// TIA Portal V19 export
VAR_GLOBAL   // PLC tag table "Digitale Eingänge"
   "E_Si_24VDC_CM01.MM01" AT %I0.0 : Bool;   // LSS 24 V OK Deckelzylinder links CM01.MM01
   "E_Si_24VDC_CM01.MM02" AT %I0.1 : Bool;   // LSS 24 V OK Deckelzylinder rechts CM01.MM02
   "E_Si_24VDC_CM02.MM03" AT %I0.2 : Bool;   // LSS 24 V OK Deckelzylinder links CM02.MM03
   "E_Si_24VDC_CM02.MM04" AT %I0.3 : Bool;   // LSS 24 V OK Deckelzylinder rechts CM02.MM04
   "R E 0.4" AT %I0.4 : Bool;
   "R E 0.5" AT %I0.5 : Bool;
   "R E 0.6" AT %I0.6 : Bool;
   E_RM_NH_Dkl AT %I0.7 : Bool;   // Rückmeldung Nothalt Deckelzylinder CM01.MM01 ... CM02.MM04
   E_Dkl_li_auf_CM01 AT %I1.0 : Bool;   // Deckel links offen int Säure CM01
   E_Dkl_li_zu_CM01 AT %I1.1 : Bool;   // Deckel links geschlossen int Säure CM01
   E_Dkl_re_auf_CM01 AT %I1.2 : Bool;   // Deckel rechts offen int Säure CM01
   E_Dkl_re_zu_CM01 AT %I1.3 : Bool;   // Deckel rechts geschlossen int Säure CM01
   "E_S_Dkl_li_auf_CM01.BG01" AT %I1.4 : Bool;   // Stellrückmeldung Deckel links offen ext CM01.BG01
   "E_S_Dkl_li_zu_CM01.BG02" AT %I1.5 : Bool;   // Stellrückmeldung Deckel links geschlossen ext CM01.BG02
   "E_S_Dkl_re_auf_CM01.BG03" AT %I1.6 : Bool;   // Stellrückmeldung Deckel rechts offen ext CM01.BG03
   "E_S_Dkl_re_zu_CM01.BG04" AT %I1.7 : Bool;   // Stellrückmeldung Deckel rechts geschlossen ext CM01.BG04
   "E_Niv_UeL_CM01.BL01" AT %I2.0 : Bool;   // Überfüllsensor Max-Max Säure CM01 CM01.BL01
   "E_Niv_Max_CM01.BL02" AT %I2.1 : Bool;   // Füllstandssensor Max Säure CM01 CM01.BL02
   "E_Niv_Min_CM01.BL03" AT %I2.2 : Bool;   // Füllstandssensor Min Säure CM01 CM01.BL03
   "E_Niv_TLS_CM01.BL04" AT %I2.3 : Bool;   // Trockenlaufschutz Min Min Säure CM01 CM01.BL04
   "E_SRM_CM01.QM25_zu" AT %I2.4 : Bool;   // Stellrückmeldung ZU Eingang Saugleitung Umwälzpumpe GP02 CM01.BG-QM25
   "E_SRM_CM01.QM18_zu" AT %I2.5 : Bool;   // Stellrückmeldung ZU Eingang Saugleitung Filterpumpe GP01 CM01.BG-QM18
   "E_SRM_CM01.QM19_zu" AT %I2.6 : Bool;   // Stellrückmeldung ZU Eingang Spülleitung Filterpumpe GP01 CM01.BG-QM19
   "E_SRM_CM01.QM20_zu" AT %I2.7 : Bool;   // Stellrückmeldung ZU Eingang Spülleitung Umwälzpumpe GP02 CM01.BG-QM20
   "E_SRM_CM01.QM26_zu" AT %I3.0 : Bool;   // Stellrückmeldung ZU Ausgang Druckleitung Umwälzpumpe GP02 CM01.BG-QM26
   "E_SRM_CM01.QM27_zu" AT %I3.1 : Bool;   // Stellrückmeldung ZU Ausgang Spülleitung Umwälzpumpe GP02 zu Sammeltank CM01.BG-QM27
   "E_GW_LF_CM01.BN01" AT %I3.2 : Bool;   // Leitfähigkeit Bypass Filterpumpe CM01.BN01
   "E_GW_LF_CM01.BN02" AT %I3.3 : Bool;   // Leitfähigkeit Düsen Umwälzung CM01.BN02
   "E_GW_p_CM01.BP03" AT %I3.4 : Bool;   // Drucksensor Filterpumpe GP01 CM01.BP03
   "E_GW_p_CM01.BP04" AT %I5.2 : Bool;   // Drucksensor Umwälzpumpe GP02 CM01.BP04
   "R E 3.6" AT %I3.6 : Bool;
   "R E 3.7" AT %I3.7 : Bool;
   "E_SRM_HQ01.QM21_auf" AT %I4.0 : Bool;   // Stellrückmeldung AUF Eingang Säureleitung Filtereinheit HQ01 HQ01.QM21
   "R E4.1" AT %I4.1 : Bool;
   "E_S_FG_li_HQ01.BG07" AT %I4.2 : Bool;   // Positionssensor Filterdeckel links HQ01 HQ01.BG07
   "E_S_FG_re_HQ01.BG08" AT %I4.3 : Bool;   // Positionssensor Filterdeckel rechts HQ01 HQ01.BG08
   "E_SRM_HQ01.QM21_zu" AT %I4.4 : Bool;   // Stellrückmeldung ZU Eingang Säureleitung Filtereinheit HQ01 HQ01.BG-QM21
   "E_SRM_HQ01.QM23_zu" AT %I4.5 : Bool;   // Stellrückmeldung ZU Ausgang Säureleitung Filtereinheit HQ01 HQ01.BG-QM23
   "E_SRM_HQ01.QM24_zu" AT %I4.6 : Bool;   // Stellrückmeldung ZU Ausgang Spülleitung Filtereinheit HQ01 zu Sammeltank HQ01.BG-QM24
   "E_SRM_HQ01.LV01_zu" AT %I4.7 : Bool;   // Stellrückmeldung ZU Entlüftungs-/Überdruckventil Beutelfilter HQ01.BG-LV01
   "E_SRM_HQ01.QM22_zu" AT %I5.0 : Bool;   // Stellrückmeldung ZU Eingang Spülleitung Filtereinheit HQ01 CM01.BG-QM22
   "E_SRM_HQ01.QM23_auf" AT %I5.1 : Bool;   // Stellrückmeldung AUF Ausgang Säureleitung Filtereinheit HQ01 HQ01.BG-QM23
   "E_GW_p_HQ01.BP01" AT %I3.5 : Bool;   // Drucksensor Beutelfiltergehäuse HQ01 HQ01.BP01
   "E_GW_p_CM03.BP05" AT %I5.3 : Bool;   // Drucksensor Umwälzpumpe GP03 CM03.BP05
   "E_Niv_Min_CM03.BL06" AT %I5.4 : Bool;   // Füllstandssensor Min Spüle CM03 CM03.BL06
   "E_Niv_TLS_CM03.BL07" AT %I5.5 : Bool;   // Trockenlaufschutz Min Min Spüle CM03 CM03.BL07
   "E_SRM_CM03.QM33_zu" AT %I5.6 : Bool;   // Stellrückmeldung ZU Eingang Saugleitung Umwälzpumpe GP03 CM03.BG-QM33
   "E_SRM_CM03.QM34_zu" AT %I5.7 : Bool;   // Stellrückmeldung ZU Ausgang Druckleitung Umwälzpumpe GP03 CM03.BG-QM34
   E_Dkl_li_auf_CM02 AT %I6.0 : Bool;   // Deckel links offen int Säure CM02
   E_Dkl_li_zu_CM02 AT %I6.1 : Bool;   // Deckel links geschlossen int Säure CM02
   E_Dkl_re_auf_CM02 AT %I6.2 : Bool;   // Deckel rechts offen int Säure CM02
   E_Dkl_re_zu_CM02 AT %I6.3 : Bool;   // Deckel rechts geschlossen int Säure CM02
   "E_S_Dkl_li_auf_CM02.BG12" AT %I6.4 : Bool;   // Stellrückmeldung Deckel links offen ext CM02.BG12
   "E_S_Dkl_li_zu_CM02.BG13" AT %I6.5 : Bool;   // Stellrückmeldung Deckel links geschlossen ext CM02.BG13
   "E_S_Dkl_re_auf_CM02.BG14" AT %I6.6 : Bool;   // Stellrückmeldung Deckel rechts offen ext CM02.BG14
   "E_S_Dkl_re_zu_CM02.BG15" AT %I6.7 : Bool;   // Stellrückmeldung Deckel rechts geschlossen ext CM02.BG15
   "E_Niv_UeL_CM02.BL08" AT %I7.0 : Bool;   // Überfüllsensor Max-Max Säure CM02 CM02.BL08
   "E_Niv_Max_CM02.BL09" AT %I7.1 : Bool;   // Füllstandssensor Max Säure CM02 CM02.BL09
   "E_Niv_Min_CM02.BL10" AT %I7.2 : Bool;   // Füllstandssensor Min Säure CM02 CM02.BL10
   "E_Niv_TLS_CM02.BL11" AT %I7.3 : Bool;   // Trockenlaufschutz Min Min Säure CM02 CM02.BL11
   "E_SRM_CM02.QM62_zu" AT %I7.4 : Bool;   // Stellrückmeldung ZU Eingang Saugleitung Umwälzpumpe GP05 CM02.BG-QM62
   "E_SRM_CM02.QM55_zu" AT %I7.5 : Bool;   // Stellrückmeldung ZU Eingang Saugleitung Filterpumpe GP04 CM02.BG-QM55
   "E_SRM_CM02.QM56_zu" AT %I7.6 : Bool;   // Stellrückmeldung ZU Eingang Spülleitung Filterpumpe GP04 CM02.BG-QM56
   "E_SRM_CM02.QM57_zu" AT %I7.7 : Bool;   // Stellrückmeldung ZU Eingang Spülleitung Umwälzpumpe GP05 CM02.BG-QM57
   "E_SRM_CM02.QM63_zu" AT %I8.0 : Bool;   // Stellrückmeldung ZU Ausgang Druckleitung Umwälzpumpe GP05 CM02.BG-QM63
   "E_SRM_CM02.QM64_zu" AT %I8.1 : Bool;   // Stellrückmeldung ZU Ausgang Spülleitung Umwälzpumpe GP05 zu Sammeltank CM02.BG-QM64
   "E_GW_LF_CM02.BN03" AT %I8.2 : Bool;   // Leitfähigkeit Bypass Filterpumpe CM02.BN03
   "E_GW_LF_CM02.BN04" AT %I8.3 : Bool;   // Leitfähigkeit Düsen Umwälzung CM02.BN04
   "E_GW_p_CM02.BP06" AT %I8.4 : Bool;   // Drucksensor Filterpumpe GP04 CM02.BP06
   "E_GW_p_HQ02.BP02" AT %I8.5 : Bool;   // Drucksensor Beutelfiltergehäuse HQ02 HQ02.BP02
   "R E 8.6" AT %I8.6 : Bool;
   "E_Niv_Uel_CM05.BL12" AT %I8.7 : Bool;   // Überfüllsensor Sammeltank CM05.BL12
   "E_LS_HQ0x.BL12" AT %I9.0 : Bool;   // Leckagesensor Filterstation HQ0x.BL12
   "R E 9.1" AT %I9.1 : Bool;
   "E_S_FG_li_HQ02.BG10" AT %I9.2 : Bool;   // Positionssensor Filterdeckel links HQ02 HQ02.BG10
   "E_S_FG_re_HQ02.BG11" AT %I9.3 : Bool;   // Positionssensor Filterdeckel rechts HQ02 HQ02.BG11
   "E_SRM_HQ02.QM59_zu" AT %I9.4 : Bool;   // Stellrückmeldung ZU Eingang Säureleitung Filtereinheit HQ02 HQ02.BG-QM59
   "E_SRM_HQ02.QM60_zu" AT %I9.5 : Bool;   // Stellrückmeldung ZU Ausgang Säureleitung Filtereinheit HQ02 HQ02.BG-QM60
   "E_SRM_HQ02.QM61_zu" AT %I9.6 : Bool;   // Stellrückmeldung ZU Ausgang Spülleitung Filtereinheit HQ02 zu Sammeltank HQ02.BG-QM61
   "E_SRM_HQ02.LV02_zu" AT %I9.7 : Bool;   // Stellrückmeldung ZU Entlüftungs-/Überdruckventil Beutelfilter HQ02.BG-LV02
   "E_SRM_HQ02.QM58_zu" AT %I10.0 : Bool;   // Stellrückmeldung ZU Eingang Spülleitung Filtereinheit HQ02 HQ02.BG-QM58
   "E_SRM_HQ01.QM24_auf" AT %I10.1 : Bool;   // Stellrückmeldung AUF Ausgang Spülleitung Filtereinheit HQ01 zu Sammeltank HQ01.BG-QM24
   "E_GW_p_CM02.BP07" AT %I10.2 : Bool;   // Drucksensor Umwälzpumpe GP05 CM02.BP07
   "E_GW_p_CM04.BP08" AT %I10.3 : Bool;   // Drucksensor Umwälzpumpe GP06 CM04.BP08
   "E_Niv_Min_CM04.BL13" AT %I10.4 : Bool;   // Füllstandssensor Min Spüle CM04 CM04.BL13
   "E_Niv_TLS_CM04.BL14" AT %I10.5 : Bool;   // Trockenlaufschutz Min Min Spüle CM04 CM04.BL14
   "E_SRM_CM04.QM72_zu" AT %I10.6 : Bool;   // Stellrückmeldung ZU Eingang Saugleitung Umwälzpumpe GP06 CM04.BG-QM72
   "E_SRM_CM04.QM73_zu" AT %I10.7 : Bool;   // Stellrückmeldung ZU Ausgang Druckleitung Umwälzpumpe GP06 CM04.BG-QM73
   E_Frg_Auto AT %I11.0 : Bool;   // Knebel Automat Ein
   "R E11.1" AT %I11.1 : Bool;   // Knebel BA Auto Reserve
   E_T_ErrQ AT %I11.2 : Bool;   // Taster Fehler Quittung
   E_T_HupeQ AT %I11.3 : Bool;   // Taster Hupe Quitt
   "R E 11.4" AT %I11.4 : Bool;   // Reserve
   "E_T_Q_Not-Halt" AT %I11.5 : Bool;   // Taster NOT-HALT Quittung Anlage
   E_T_Frg_BE AT %I11.6 : Bool;   // Quittierschalter Beizkorb einfahren/holen Be-/Entladestation WR01 WR01.SF01
   "E_LS_CL01.BL28" AT %I11.7 : Bool;   // Leckage OK Übergabestation CL01 CL01.BL28
   "E_LS_CL02.BL29" AT %I12.0 : Bool;   // Leckage OK Pumpensumpf Säurebecken CL02 CL02.BL29
   "E_GW_p_CM05.BP09" AT %I12.1 : Bool;   // Drucksensor Entleerung Sammeltank CM05 CM05.BP09
   "E_Niv_max_CM05.BL01" AT %I12.2 : Bool;   // Vollmeldung Sammeltank CM05 CM05.BL01
   "E_Niv_min_CM05.BL02" AT %I12.3 : Bool;   // Leermeldung Sammeltank CM05 CM05.BL02
   "E_Niv_TLS_CM05.BL03" AT %I12.4 : Bool;   // Trockenlaufschutz Sammeltank CM05 CM05.BL03
   "E_SRM_CM05.QM61_zu" AT %I12.5 : Bool;   // Stellrückmeldung ZU Absperrventil Saugseite Förderpumpe GP11 CM05.BG-QM61
   "E_SRM_CM05.QM64_zu" AT %I12.6 : Bool;   // Stellrückmeldung ZU Absperrventil Druckseite Förderpumpe GP11 CM05.BG-QM64
   "E_Normal-Vers" AT %I12.7 : Bool;   // Normalversorgung aktiv
   "E_Not-Strom" AT %I13.0 : Bool;   // Notstromversorgung aktiv
   E_Frg_AbLW AT %I13.1 : Bool;   // Abluftwäscher OK (Freigabe)
   E_Wrn_Gas_ok AT %I13.2 : Bool;   // Gaswarnanlage Voralarm
   E_Al_Gas_ok AT %I13.3 : Bool;   // Gaswarnanlage Hauptalarm
   E_AWA_ok AT %I13.4 : Bool;   // Neutralisation betriebsbereit
   E_Frg_AWA AT %I13.5 : Bool;   // Freigabe Abpumpen von Neutralisation
   E_kein_NB_AblW AT %I13.6 : Bool;   // Kein Notbetrieb Abluftwäscher
   E_VEW_ok AT %I13.7 : Bool;   // Druck VE-Wasser o.k.
   E_DL_min_ok AT %I14.0 : Bool;   // Druckluft > 5.0 bar
   E_DL_keine_Warnung AT %I14.1 : Bool;   // Druckluft > 5.3 bar
   E_StrWae_Abluft_ok AT %I14.2 : Bool;   // Strömungswächter Abluftleitung o.k.
   E_UeSp_ok AT %I14.3 : Bool;   // Überspannungsableiter OK
   E_Si_230VAC_Bel AT %I14.4 : Bool;   // LSS OK Beleuchtung im Tunnel FP02.GQ01
   "R E 14.5" AT %I14.5 : Bool;
   "R E 14.6" AT %I14.6 : Bool;
   "R E 14.7" AT %I14.7 : Bool;
   E_MSS_ok_RT AT %I15.0 : Bool;   // MSS OK Schnelllauftor Ein-/Ausfahrt
   E_S_RT_auf AT %I15.1 : Bool;   // Schnelllauftor offen Ein-/Ausfahrt
   E_S_RT_zu AT %I15.2 : Bool;   // Schnelllauftor geschlossen Ein-/Ausfahrt
   E_RT_ok AT %I15.3 : Bool;   // Schnelllauftor OK Ein-/Ausfahrt
   "E_MSS_ok_CM05.GP11" AT %I15.4 : Bool;   // MSS OK Pumpe Entleerung Sammeltank CM05.GP11
   "E_RM_NH_FP_CM01.GP01" AT %I15.5 : Bool;   // Rückmeldung Nothalt Filterpumpen CM01.GP01
   "E_RM_NH_FP_CM01.GP04" AT %I15.6 : Bool;   // Rückmeldung Nothalt Filterpumpen CM02.GP04
   E_RM_NH_Pumpen AT %I15.7 : Bool;   // Rückmeldung Nothalt Pumpen
   "E_SRM_CM01.QM25_auf" AT %I16.0 : Bool;   // Stellrückmeldung AUF Eingang Saugleitung Umwälzpumpe GP02 CM01.BG-QM25
   "E_SRM_CM01.QM18_auf" AT %I16.1 : Bool;   // Stellrückmeldung AUF Eingang Saugleitung Filterpumpe GP01 CM01.BG-QM18
   "E_SRM_CM01.QM19_auf" AT %I16.2 : Bool;   // Stellrückmeldung AUF Eingang Spülleitung Filterpumpe GP01 CM01.BG-QM19
   "E_SRM_CM01.QM20_auf" AT %I16.3 : Bool;   // Stellrückmeldung AUF Eingang Spülleitung Umwälzpumpe GP02 CM01.BG-QM20
   "E_SRM_CM01.QM26_auf" AT %I16.4 : Bool;   // Stellrückmeldung AUF Ausgang Druckleitung Umwälzpumpe GP02 CM01.BG-QM26
   "E_SRM_CM01.QM27_auf" AT %I16.5 : Bool;   // Stellrückmeldung AUF Ausgang Spülleitung Umwälzpumpe GP02 zu Sammeltank CM01.BG-CM01.QM27
   "E_SRM_CM03.QM33_auf" AT %I16.6 : Bool;   // Stellrückmeldung AUF Eingang Saugleitung Umwälzpumpe GP03 CM03.BG-QM33
   "E_SRM_CM03.QM34_auf" AT %I16.7 : Bool;   // Stellrückmeldung AUF Ausgang Druckleitung Umwälzpumpe GP03 CM03.BG-QM34
   "E_SRM_CM02.QM62_auf" AT %I17.0 : Bool;   // Stellrückmeldung AUF Eingang Saugleitung Umwälzpumpe GP05 CM02.BG-QM62
   "E_SRM_CM02.QM55_auf" AT %I17.1 : Bool;   // Stellrückmeldung AUF Eingang Saugleitung Filterpumpe GP04 CM02.BG-QM55
   "E_SRM_CM02.QM56_auf" AT %I17.2 : Bool;   // Stellrückmeldung AUF Eingang Spülleitung Filterpumpe GP04 CM02.BG-QM56
   "E_SRM_CM02.QM57_auf" AT %I17.3 : Bool;   // Stellrückmeldung AUF Eingang Spülleitung Umwälzpumpe GP05 CM02.BG-QM57
   "E_SRM_CM02.QM63_auf" AT %I17.4 : Bool;   // Stellrückmeldung AUF Ausgang Druckleitung Umwälzpumpe GP05 CM02.BG-QM63
   "E_SRM_CM02.QM64_auf" AT %I17.5 : Bool;   // Stellrückmeldung AUF Ausgang Spülleitung Umwälzpumpe GP05 zu Sammeltank CM02.BG-CM02.QM64
   "E_SRM_HQ01.LV01_auf" AT %I17.6 : Bool;   // Stellrückmeldung AUF Entlüftungs-/Überdruckventil Beutelfilter HQ01.BG-LV01
   "E_SRM_HQ01.QM22_auf" AT %I17.7 : Bool;   // Stellrückmeldung AUF Eingang Spülleitung Filtereinheit HQ01 HQ01.BG-QM22
   "E_LS_GP01.BL15" AT %I32.0 : Bool;   // Membran-Leckagesensor Pumpe GP13 Versorgung Frischsäure GP01.BL15
   "E_LS_GP01.BL16" AT %I32.1 : Bool;   // Leckagesensor PFA-Übergang auf GP01 Dopelrohrleitung GP01.BL16
   "E_Niv_min_GP01.BL17" AT %I32.2 : Bool;   // Leermeldung Gebinde HF IBC Sauglanze GP01.BL17
   "E_Niv_max_GP01.BL20" AT %I32.3 : Bool;   // IBC-Füllstand voll Gebinde HF IBC Versorgung Frischsäure GP01.BL20
   "E_S_IBC_GP01.BG21" AT %I32.4 : Bool;   // IBC-Erkennung Gebinde HF IBC Versorgung Frischsäure GP01.BG21
   "R E 32.5" AT %I32.5 : Bool;
   "R E 32.6" AT %I32.6 : Bool;
   "E_LS_GP01.BL18" AT %I32.7 : Bool;   // Leckage OK Pumpensumpf Versorgung GP01 GP01.BL18
   "E_LS_GP01.BL19" AT %I33.0 : Bool;   // Leckagesensor Verteiler GP01 Doppelrohrleitung GP01.BL19 (UV)
   "E_SRM_GP01.QM15_zu" AT %I33.1 : Bool;   // Stellrückmeldung ZU Eingang Saugleitung Membranpumpe GP13 GP01.BG-QM15
   "E_SRM_GP01.QM16_zu" AT %I33.2 : Bool;   // Stellrückmeldung ZU Eingang Spülleitung Membranpumpe GP13 GP01.BG-QM16
   "E_SRM_GP01.QM17_zu" AT %I33.3 : Bool;   // Stellrückmeldung ZU Ausgang Spülleitung Membranpumpe GP13 GP01.BG-QM17
   "E_SRM_GP01.QM18_zu" AT %I33.4 : Bool;   // Stellrückmeldung ZU Ausgang Druckleitung Membranp. GP13 zu UV-GP01 GP01.BG-QM18
   "E_SRM_GP01.QM19_zu" AT %I33.5 : Bool;   // Stellrückmeldung ZU Verriegelung UV-GP01 Versorgungsleitung zu CM02 GP01.BG-QM19
   "E_SRM_GP01.QM20_zu" AT %I33.6 : Bool;   // Stellrückmeldung ZU Verriegelung UV-GP01 Versorgungsleitung zu CM01 GP01.BG-QM20
   "E_SRM_GP01.QM21_zu" AT %I33.7 : Bool;   // Stellrückmeldung ZU Verriegelung UV-GP01 Versorgungsleitung zu GP02 GP01.BG-QM21
   "E_SRM_GP01.QM22_zu" AT %I34.0 : Bool;   // Stellrückmeldung ZU Verriegelung UV-GP01 Versorgungsl. zu GP01 GP01.BG-QM22
   "E_Imp_GP01.BF01" AT %I34.1 : Bool;   // Durchfluss-Impuls Versorgung Frischsäure GP01 GP01.BF01
   "E_GW_Dfl_GP01.BF01" AT %I34.2 : Bool;   // Durchfluss-Leerrohr Versorgung Frischsäure GP01 GP01.BF01
   "E_LS_GP01.BL34" AT %I34.3 : Bool;   // Leckage Umleitung zum Tunnel (von Versorgung GP01)
   "E_LS_GP02.BL32" AT %I34.4 : Bool;   // Leckagesensor Doppelschlauch zur Versorgung GP02 --> UV GP01
   "E_LS_GP02.BL33" AT %I34.5 : Bool;   // Leckagesensor Doppelschlauch zu Entsorgung GP02
   "R E34.6" AT %I34.6 : Bool;
   "R E34.7" AT %I34.7 : Bool;
   "E_LS_GP02.BL27" AT %I35.0 : Bool;   // Membran-Leckagesensor Pumpe GP10 Entsorgung Altsäure GP02.BL27
   "E_S_IBC_GP02.BG22" AT %I35.1 : Bool;   // IBC-Erkennung Gebinde HF IBC Versorgung Frischsäure GP02.BG22
   "E_Niv_max_GP02.BL23" AT %I35.2 : Bool;   // IBC-Füllstand voll Gebinde HF IBC Versorgung Frischsäure GP02.BL23
   "E_Niv_min_GP02.BL24" AT %I35.3 : Bool;   // Leermeldung Gebinde HF IBC Sauglanze GP02.BL24
   "E_SRM_GP02.QM38_zu" AT %I35.4 : Bool;   // Stellrückmeldung ZU Eingang Saugleitung Membranpumpe GP10 GP02.BG-QM38
   "R E 35.5" AT %I35.5 : Bool;
   "E_SRM_GP02.QM38_auf" AT %I35.6 : Bool;   // Stellrückmeldung AUF Eingang Saugleitung Membranpumpe GP10 GP02.BG-QM38
   "E_LS_GP02.BL21" AT %I35.7 : Bool;   // Leckage OK Pumpensumpf Entsorgung GP02 GP02.BL21
   "E_LS_GP02.BL26" AT %I36.0 : Bool;   // Leckagesensor Verteiler GP02 Doppelrohrleitung GP02.BL26 (UV)
   "E_SRM_GP02.QM39_zu" AT %I36.1 : Bool;   // Stellrückmeldung ZU Eingang Spülleitung Membranpumpe GP10 GP02.BG-QM39
   "E_SRM_GP02.QM40_zu" AT %I36.2 : Bool;   // Stellrückmeldung ZU Ausgang Druckleitung Membranpumpe GP10 GP02.BG-QM40
   "E_SRM_GP02.QM41_zu" AT %I36.3 : Bool;   // Stellrückmeldung ZU Verriegelung UV-GP02 Versorgungsleitung zu GP02 GP02.BG-QM41
   "E_SRM_GP02.QM42_zu" AT %I36.4 : Bool;   // Stellrückmeldung ZU Ausgang Spülleitung Membranpumpe GP10 zu CM05 GP02.BG-QM42
   "R E 36.5" AT %I36.5 : Bool;
   "R E 36.6" AT %I36.6 : Bool;
   "E_SRM_GP02.QM45_zu" AT %I36.7 : Bool;   // Stellrückmeldung ZU Verriegelung UV-GP02 Entsorgungsleitung von CM01 GP02.BG-QM45
   "E_SRM_GP02.QM46_zu" AT %I37.0 : Bool;   // Stellrückmeldung ZU Verriegelung UV-GP02 Entsorgungsleitung von CM02 GP02.BG-QM46
   "E_Imp_GP02.BF02" AT %I37.1 : Bool;   // Durchfluss-Impuls Entsorgung Altsäure GP02 GP02.BF02
   "E_GW_Dfl_GP02.BF02" AT %I37.2 : Bool;   // Durchfluss-Leerrohr Entsorgung Altsäure GP02 GP02.BF02
   "E_SRM_GP01.QM15_auf" AT %I37.3 : Bool;   // Stellrückmeldung AUF Eingang Saugleitung Membranpumpe GP13 GP01.BG-QM15
   "E_SRM_GP01.QM16_auf" AT %I37.4 : Bool;   // Stellrückmeldung AUF Eingang Spülleitung Membranpumpe GP13 GP01.BG-QM16
   "E_SRM_GP01.QM17_auf" AT %I37.5 : Bool;   // Stellrückmeldung AUF Ausgang Spülleitung Membranpumpe GP13 GP01.BG-QM17
   "E_SRM_GP01.QM18_auf" AT %I37.6 : Bool;   // Stellrückmeldung AUF Ausgang Druckleitung Membranp. GP13 zu UV-GP01 GP01.BG-QM18
   "E_LS_GP02.BL25" AT %I37.7 : Bool;   // Leckagesensor PFA-Übergang auf GP02 Dopelrohrleitung GP02.BL25
   "E_SRM_HQ02.QM59_auf" AT %I18.0 : Bool;   // Stellrückmeldung AUF Eingang Säureleitung Filtereinheit HQ02 HQ02.BG-QM59
   "E_SRM_HQ02.QM60_auf" AT %I18.1 : Bool;   // Stellrückmeldung AUF Ausgang Säureleitung Filtereinheit HQ02 HQ02.BG-QM60
   "E_SRM_HQ02.QM61_auf" AT %I18.2 : Bool;   // Stellrückmeldung AUF Ausgang Spülleitung Filtereinheit HQ02 zu Sammeltank HQ02.BG-HQ02.QM61
   "E_SRM_HQ02.LV02_auf" AT %I18.3 : Bool;   // Stellrückmeldung AUF Entlüftungs-/Überdruckventil Beutelfilter HQ02.BG-LV02
   "E_SRM_HQ02.QM58_auf" AT %I18.4 : Bool;   // Stellrückmeldung AUF Eingang Spülleitung Filtereinheit HQ02 HQ02.BG-QM58
   "E_SRM_CM04.QM72_auf" AT %I18.5 : Bool;   // Stellrückmeldung AUF Eingang Saugleitung Umwälzpumpe GP06 CM04.BG-QM72
   "E_SRM_CM04.QM73_auf" AT %I18.6 : Bool;   // Stellrückmeldung AUF Ausgang Druckleitung Umwälzpumpe GP06 CM04.BG-QM73
   "E_SRM_CM05.QM61_auf" AT %I18.7 : Bool;   // Stellrückmeldung AUF Absperrventil Saugseite Förderpumpe GP11 CM05.BG-QM61
   "E_SRM_CM05.QM64_auf" AT %I19.0 : Bool;   // Stellrückmeldung AUF Absperrventil Druckseite Förderpumpe GP11 CM05.BG-QM64
   "R E 19.1" AT %I19.1 : Bool;
   "R E 19.2" AT %I19.2 : Bool;
   "R E 19.3" AT %I19.3 : Bool;
   "R E 19.4" AT %I19.4 : Bool;
   "R E 19.5" AT %I19.5 : Bool;
   "R E 19.6" AT %I19.6 : Bool;
   "R E 19.7" AT %I19.7 : Bool;
   "E_SRM_GP01.QM19_auf" AT %I38.0 : Bool;   // Stellrückmeldung AUF Verriegelung UV-GP01 Versorgungsleitung zu CM02 GP01.BG-QM1
   "E_SRM_GP01.QM20_auf" AT %I38.1 : Bool;   // Stellrückmeldung AUF Verriegelung UV-GP01 Versorgungsleitung zu CM01 GP01.BG-QM2
   "E_SRM_GP01.QM21_auf" AT %I38.2 : Bool;   // Stellrückmeldung AUF Verriegelung UV-GP01 Versorgungsleitung zu GP02 GP01.BG-QM2
   "E_SRM_GP01.QM22_auf" AT %I38.3 : Bool;   // Stellrückmeldung AUF Verriegelung UV-GP01 Versorgungsl. zu GP01 GP01.BG-QM22
   "E_SRM_GP02.QM39_auf" AT %I38.4 : Bool;   // Stellrückmeldung AUF Eingang Spülleitung Membranpumpe GP10 GP02.BG-QM39
   "E_SRM_GP02.QM40_auf" AT %I38.5 : Bool;   // Stellrückmeldung AUF Ausgang Druckleitung Membranpumpe GP10 GP02.BG-QM40
   "E_SRM_GP02.QM41_auf" AT %I38.6 : Bool;   // Stellrückmeldung AUF Verriegelung UV-GP02 Versorgungsleitung zu GP02 GP02.BG-QM41
   "E_SRM_GP02.QM42_auf" AT %I38.7 : Bool;   // Stellrückmeldung AUF Ausgang Spülleitung Membranpumpe GP10 zu CM05 GP02.BG-QM42
   "R E 39.0" AT %I39.0 : Bool;
   "R E 39.1" AT %I39.1 : Bool;
   "E_SRM_GP02.QM45_auf" AT %I39.2 : Bool;   // Stellrückmeldung AUF Verriegelung UV-GP02 Entsorgungsleitung von CM01 GP02.BG-QM45
   "E_SRM_GP02.QM46_auf" AT %I39.3 : Bool;   // Stellrückmeldung AUF Verriegelung UV-GP02 Entsorgungsleitung von CM02 GP02.BG-QM46
   "E_SRM_GP01.QM14_zu" AT %I39.4 : Bool;
   "E_SRM_GP01.QM14_auf" AT %I39.5 : Bool;
   "R E 39.6" AT %I39.6 : Bool;
   "R E 39.7" AT %I39.7 : Bool;
   "R E 72.0" AT %I72.0 : Bool;
   "R E 72.1" AT %I72.1 : Bool;
   "R E 72.2" AT %I72.2 : Bool;
   "R E 72.3" AT %I72.3 : Bool;
   E_S_vl_QF1_frei AT %I72.4 : Bool;   // Querumsetzer 1 Sensor Beizkorberkennung Auflage vorne links WR02.BG17
   E_S_vr_QF1_frei AT %I72.5 : Bool;   // Querumsetzer 1 Sensor Beizkorberkennung Auflage vorne rechts WR02.BG18
   E_S_hl_QF1_frei AT %I72.6 : Bool;   // Querumsetzer 1 Sensor Beizkorberkennung Auflage hinten links WR02.BG19
   E_S_hr_QF1_frei AT %I72.7 : Bool;   // Querumsetzer 1 Sensor Beizkorberkennung Auflage hinten rechts WR02.BG20
   E_S_Pos_BE_QF1 AT %I73.0 : Bool;   // Querumsetzer 1 Sensor Endlage Beladestation WR02.BG16
   E_S_lgsm_to_BE_QF1 AT %I73.1 : Bool;   // Querumsetzer 1 Sensor langsam Beladestation WR02.BG21
   E_S_lgsm_to_Ue_QF1 AT %I73.2 : Bool;   // Querumsetzer 1 Sensor langsam Übergabestation WR02.BG22
   E_S_Pos_Ue_QF1 AT %I73.3 : Bool;   // Querumsetzer 1 Sensor Endlage Übergabestation WR02.BG23
   E_S_vl_QF2_frei AT %I73.4 : Bool;   // Querumsetzer 2 Sensor Beizkorberkennung Auflage vorne links WR03.BG23
   E_S_vr_QF2_frei AT %I73.5 : Bool;   // Querumsetzer 2 Sensor Beizkorberkennung Auflage vorne rechts WR03.BG24
   E_S_hl_QF2_frei AT %I73.6 : Bool;   // Querumsetzer 2 Sensor Beizkorberkennung Auflage hinten links WR03.BG25
   E_S_hr_QF2_frei AT %I73.7 : Bool;   // Querumsetzer 2 Sensor Beizkorberkennung Auflage hinten rechts WR03.BG26
   E_S_Pos_BE_QF2 AT %I74.0 : Bool;   // Querumsetzer 2 Sensor Endlage Beladestation WR03.BG22
   E_S_lgsm_to_BE_QF2 AT %I74.1 : Bool;   // Querumsetzer 2 Sensor langsam Beladestation WR03.BG27
   E_S_lgsm_to_Ue_QF2 AT %I74.2 : Bool;   // Querumsetzer 2 Sensor langsam Übergabestation WR03.BG28
   E_S_Pos_Ue_QF2 AT %I74.3 : Bool;   // Querumsetzer 2 Sensor Endlage Übergabestation WR03.BG29
   "R E 74.4" AT %I74.4 : Bool;
   "R E 74.5" AT %I74.5 : Bool;
   "R E 74.6" AT %I74.6 : Bool;
   "R E 74.7" AT %I74.7 : Bool;
   "R E 75.0" AT %I75.0 : Bool;
   "R E 75.1" AT %I75.1 : Bool;
   "R E 75.2" AT %I75.2 : Bool;
   "R E 75.3" AT %I75.3 : Bool;
   "R E 75.4" AT %I75.4 : Bool;
   "R E 75.5" AT %I75.5 : Bool;
   "R E 75.6" AT %I75.6 : Bool;
   "R E 75.7" AT %I75.7 : Bool;
   E_BE_vor_TW AT %I80.0 : Bool;   // Manipulator Sensor Notendlage vorwärts WR04.BG42
   E_BE_rck_TW AT %I80.1 : Bool;   // Manipulator Sensor Notendlage rückwärts WR04.BG43
   E_Not_oben_re AT %I80.2 : Bool;   // Hubwerk rechts Sensor Notendlage oben WR04.BG28
   E_not_unten_re AT %I80.3 : Bool;   // Hubwerk rechts Sensor Notendlage unten WR04.BG29
   E_GurtUeL_re AT %I80.4 : Bool;   // Hubwerk rechts Bandüberlauf WR04.BG32
   "R E80.5" AT %I80.5 : Bool;
   E_UeL_ok_re AT %I80.6 : Bool;   // Hubwerk rechts Störung/Überlast Lastmessbolzen WR04.BW34
   E_Frg_Snk_re AT %I80.7 : Bool;   // Hubwerk rechts Freigabe Senken Lastmessbolzen WR04.BW34
   E_Frg_Heb_re AT %I81.0 : Bool;   // Hubwerk rechts Freigabe Heben Lastmessbolzen WR04.BW34
   E_WZ_ok_re_1 AT %I81.1 : Bool;   // Hubwerk rechts Wägezelle 1 OK WR04.BW01
   E_WZ_ok_re_2 AT %I81.2 : Bool;   // Hubwerk rechts Wägezelle 2 OK WR04.BW02
   E_WZ_ok_re_3 AT %I81.3 : Bool;   // Hubwerk rechts Wägezelle 3 OK WR04.BW03
   E_WZ_ok_re_4 AT %I81.4 : Bool;   // Hubwerk rechts Wägezelle 4 OK WR04.BW04
   "R E 81.5" AT %I81.5 : Bool;
   "R E 81.6" AT %I81.6 : Bool;
   "R E 81.7" AT %I81.7 : Bool;
   "R E 82.0" AT %I82.0 : Bool;
   "R E 82.1" AT %I82.1 : Bool;
   E_Not_oben_li AT %I82.2 : Bool;   // Hubwerk links Sensor Notendlage oben WR05.BG36
   E_not_unten_li AT %I82.3 : Bool;   // Hubwerk links Sensor Notendlage unten WR05.BG37
   E_GurtUeL_li AT %I82.4 : Bool;   // Hubwerk links Bandüberlauf WR05.BG39
   "R E82.5" AT %I82.5 : Bool;
   E_UeL_ok_li AT %I82.6 : Bool;   // Hubwerk links Störung/Überlast Lastmessbolzen WR05.BW43
   E_Frg_Snk_li AT %I82.7 : Bool;   // Hubwerk links Freigabe Senken Lastmessbolzen WR05.BW43
   E_Frg_Heb_li AT %I83.0 : Bool;   // Hubwerk links Freigabe Heben Lastmessbolzen WR05.BW43
   E_WZ_ok_li_1 AT %I83.1 : Bool;   // Hubwerk links Wägezelle 1 OK WR05.BW01
   E_WZ_ok_li_2 AT %I83.2 : Bool;   // Hubwerk links Wägezelle 2 OK WR05.BW02
   E_WZ_ok_li_3 AT %I83.3 : Bool;   // Hubwerk links Wägezelle 3 OK WR05.BW03
   E_WZ_ok_li_4 AT %I83.4 : Bool;   // Hubwerk links Wägezelle 4 OK WR05.BW04
   "R E 83.5" AT %I83.5 : Bool;
   "R E 83.6" AT %I83.6 : Bool;
   "R E 83.7" AT %I83.7 : Bool;
   ED_PosInc_348i_TW AT %ID310 : DInt;   // Incremente Fahrt TW
   EW_Status_348i_TW AT %IW314 : Word;   // Status Laser TW
   ED_HubInc_li_TW AT %ID320 : DInt;   // Incremente Hub links
   ED_HubInc_re_TW AT %ID330 : DInt;   // Incremente Hub rechts
   EB_RM_StB_Preset_SL_links AT %IB324 : Byte;
   EB_RM_StB_Preset_SL_rechts AT %IB334 : Byte;
END_VAR
